ABB RAPID module: Wobj_FRAME_PalletEntrada.mod

MODULE Wobj_FRAME_PalletEntrada
	! Points are read in order of declaration.
  ! Please do not change the order of points!

  LOCAL PERS robtarget pWobj_U_PointX1:=[[-2197.262,1272.152,425.5257],[0.285739362239838,-0.921125411987305,0.263248473405838,0.0241078287363052],[1,-1,0,0],[9E+09,9E+09,9E+09,9E+09,9E+09,9E+09]];
	LOCAL PERS robtarget pWobj_U_PointX2:=[[-2209.013,1998.444,431.8939],[0.285738527774811,-0.921125113964081,0.263251066207886,0.0241009593009949],[1,-1,0,0],[9E+09,9E+09,9E+09,9E+09,9E+09,9E+09]];
	LOCAL PERS robtarget pWobj_U_PointY1:=[[-2687.02,1266.622,426.6517],[0.285737544298172,-0.92112672328949,0.263245642185211,0.0241114944219589],[1,-1,0,0],[9E+09,9E+09,9E+09,9E+09,9E+09,9E+09]];

ENDMODULE
